FUNCTION_BLOCK FB_MatrixShrink_Test EXTENDS FB_TestSuite
VAR_INPUT
END_VAR
VAR_OUTPUT
END_VAR
VAR
END_VAR

WhenEmptyExpectError();
WhenShrunkExpectDataRetained();

METHOD PRIVATE WhenEmptyExpectError
VAR_INPUT
END_VAR
VAR
	M1 : Matrix;
	M2 : Matrix;
	Result : BOOL;
END_VAR
TEST('WhenEmptyExpectError');

// @TEST-RUN
M1.InitZeros(1,1);
Result := M2.AsShrunk(M1,0,0);

// @TEST-ASSERT
AssertFalse(Result,'Main function call was unexpectedly successful');

TEST_FINISHED();
END_METHOD

METHOD PRIVATE WhenShrunkExpectDataRetained
VAR_INPUT
END_VAR
VAR
	M1 : Matrix;
	M2 : Matrix;
	M3 : Matrix;
	Result : BOOL;
END_VAR
TEST('WhenShrunkExpectDataRetained');

// @TEST-RUN
M1.InitMagicSquare(3);
Result := M2.AsShrunk(M1,0,0);
M3.AsSubMatrix(M1,1,2,1,2);

// @TEST-ASSERT
AssertTrue(Result,'Main function call was not successful');
AssertTrue(M3.IsEqual(M2),'Old data was not retained');

TEST_FINISHED();
END_METHOD

END_FUNCTION_BLOCK

(* stored: Version 1.1.0.1, ProductVersion 3.1.4024.9
   POU FB_MatrixShrink_Test: Id {6badab89-4b35-0a67-0e21-0fcc6b60e2f9}, SpecialFunc None
   Method WhenEmptyExpectError: Id {d6787aff-e80e-04a9-15be-66639abd753f}
   Method WhenShrunkExpectDataRetained: Id {a2dd6e96-bc8c-06dc-0aa7-16350c013705} *)
